// TIA Portal V17 export
// export: Created 2022-07-20T06:59:48.1085012Z, ExportSetting WithDefaults, DisplayName Totally Integrated Automation Portal, DisplayVersion V17, DisplayName TIA Portal Openness, DisplayVersion V17, DisplayName TIA Portal Version Control Interface, DisplayVersion V17, DisplayName SINAMICS Startdrive Advanced, DisplayVersion V17, DisplayName SINAMICS Startdrive G130, G150, S120, S150, SINAMICS MV, S210, DisplayVersion V17, DisplayName SINAMICS Startdrive G110M, G120, G120C, G120D, G120P, G115D, DisplayVersion V17, DisplayName STEP 7 Professional, DisplayVersion V17, DisplayName STEP 7 Safety, DisplayVersion V17, DisplayName WinCC Advanced, DisplayVersion V17
FUNCTION_BLOCK "FB10191_SheetTrackingProcess"   // FB10191, LAD
{ S7_Optimized_Access := 'TRUE' }
VERSION : 0.1
// stored: AutoNumber false, IsIECCheckEnabled false, IsRetainMemResEnabled false, MemoryReserve 100, SetENOAutomatically false, UDAEnableTagReadback false
   VAR_INPUT
      Enable : Bool;
      FirstSheetSensor : Bool;
      SecondSheetSensor : Bool;
      SheetSize : Real;   // mm
      TransportSpeed : Real;   // mm/s
      ActivationProcessMargin : Real;   // 0-100%
      DeactivationProcessMargin : Real;
      DistanceBetweenSheetSensors : Real;
      DistanceBetweenSheetSensorAndProcess : Real;
      RequestAcknowledge : Bool;
      Reset : Bool;
   END_VAR
   VAR_OUTPUT
      ActiveProcess : Bool;
      DeactiveProcess : Bool;
      TrackingProcessInError : Bool;
   END_VAR
   VAR
      i : SInt;
      R_TRIG_Enable : R_TRIG;
      R_TRIG_Reset { S7_SetPoint := 'True'} : R_TRIG;
      R_TRIG_Clock10Hz : R_TRIG;
      R_TRIG_SheetSensorSignal_1 { S7_SetPoint := 'True'} : R_TRIG;
      R_TRIG_SheetSensorSignal_2 { S7_SetPoint := 'True'} : R_TRIG;
      R_TRIG_SheetOutsideProcess { S7_SetPoint := 'True'} : R_TRIG;
      F_TRIG_Enable { S7_SetPoint := 'True'} : F_TRIG;
      F_TRIG_Clock10Hz { S7_SetPoint := 'True'} : F_TRIG;
      F_TRIG_SheetSensorSignal_1 { S7_SetPoint := 'True'} : F_TRIG;
      F_TRIG_SheetSensorSignal_2 { S7_SetPoint := 'True'} : F_TRIG;
      ARRAY_R_TRIGS_SheetsSensor_1 : Array[0..49] of Bool;
      ARRAY_R_TRIGS_SheetsSensor_2 : Array[0..49] of Bool;
      ARRAY_R_TRIGS_BeginningOfSheetUnderProcess : Array[0..49] of R_TRIG;
      ARRAY_R_TRIGS_EndOfSheetUnderProcess : Array[0..49] of R_TRIG;
      ARRAY_F_TRIGS_SheetsSensor_1 : Array[0..49] of Bool;
      ARRAY_F_TRIGS_SheetsSensor_2 : Array[0..49] of Bool;
      ARRAY_BeginingOfSheetPosition { S7_SetPoint := 'True'} : Array[0..49] of Real;   // mm
      ARRAY_EndOfSheetPosition { S7_SetPoint := 'True'} : Array[0..49] of Real;   // mm
      ARRAY_ElpasedTimeFromPreviousCheck { S7_SetPoint := 'True'} : Array[0..49] of Time;   // s
      ARRAY_TON_SheetsBetweenSensors : Array[0..49] of TON_TIME;
   END_VAR
BEGIN

REGION Network 1 (SCL): First Scan & Reset
   IF "FirstScan" OR #R_TRIG_Enable.Q OR #F_TRIG_Enable.Q OR #R_TRIG_Reset.Q THEN
       #ActiveProcess := FALSE;
       #DeactiveProcess := TRUE;
       FOR #i := 0 TO 49 DO
           #ARRAY_R_TRIGS_SheetsSensor_1[#i] := FALSE;
           #ARRAY_F_TRIGS_SheetsSensor_1[#i] := FALSE;
           #ARRAY_R_TRIGS_SheetsSensor_2[#i] := FALSE;
           #ARRAY_F_TRIGS_SheetsSensor_2[#i] := FALSE;
           #ARRAY_BeginingOfSheetPosition[#i] := 0.0;
           #ARRAY_EndOfSheetPosition[#i] := 0.0;
           #ARRAY_ElpasedTimeFromPreviousCheck[#i] := T#0s;
           RESET_TIMER(#ARRAY_TON_SheetsBetweenSensors[#i]);
       END_FOR;
   END_IF;
END_REGION

REGION Network 2 (SCL): Edge Signals & Timers
   REGION EDGE SIGNALS
       #R_TRIG_Enable(CLK := #Enable);
       #R_TRIG_Reset(CLK := #Reset);

       #F_TRIG_Enable(CLK := #Enable);
   END_REGION

   IF #Enable THEN
       REGION EDGE SIGNALS
           #R_TRIG_Clock10Hz(CLK := "Clock_10Hz");
           #R_TRIG_SheetSensorSignal_1(CLK := #FirstSheetSensor);
           #R_TRIG_SheetSensorSignal_2(CLK := #SecondSheetSensor);
           #R_TRIG_SheetOutsideProcess(CLK :=
                                       (#ARRAY_R_TRIGS_SheetsSensor_1[0] AND
                                       #ARRAY_R_TRIGS_SheetsSensor_2[0] AND
                                       #ARRAY_F_TRIGS_SheetsSensor_1[0] AND
                                       #ARRAY_F_TRIGS_SheetsSensor_2[0])
                                       OR
                                       (#ARRAY_BeginingOfSheetPosition[0] > 2 * #DistanceBetweenSheetSensors));

           #F_TRIG_Clock10Hz(CLK := "Clock_10Hz");
           #F_TRIG_SheetSensorSignal_1(CLK := #FirstSheetSensor);
           #F_TRIG_SheetSensorSignal_2(CLK := #SecondSheetSensor);

           FOR #i := 0 TO 49 DO
               #ARRAY_R_TRIGS_BeginningOfSheetUnderProcess[#i](CLK := #ARRAY_R_TRIGS_SheetsSensor_1[#i] AND "FC10021_TolerenceRelation"(X := #ARRAY_BeginingOfSheetPosition[#i], Y := #DistanceBetweenSheetSensorAndProcess, Tolerance := ((1 + #ActivationProcessMargin / 100) * 100)));
               #ARRAY_R_TRIGS_EndOfSheetUnderProcess[#i](CLK := #ARRAY_F_TRIGS_SheetsSensor_1[#i] AND "FC10021_TolerenceRelation"(X := #ARRAY_EndOfSheetPosition[#i], Y := #DistanceBetweenSheetSensorAndProcess, Tolerance := ((1 + #DeactivationProcessMargin / 100) * 100)));
           END_FOR;
       END_REGION

       REGION TIMERS
           FOR #i := 0 TO 49 DO
               #ARRAY_TON_SheetsBetweenSensors[#i](IN := #ARRAY_R_TRIGS_SheetsSensor_1[#i] AND NOT (#ARRAY_F_TRIGS_SheetsSensor_2[#i]),
                                                   PT := DINT_TO_TIME(REAL_TO_DINT((1 + (#ActivationProcessMargin / 100.0)) * (#DistanceBetweenSheetSensors / #TransportSpeed)) * 1000));
           END_FOR;
       END_REGION
   END_IF;
END_REGION

REGION Network 3 (SCL): Sheet Position Management
   IF #Enable THEN
      //Detect to Rising Edge of the first sensor
       IF #R_TRIG_SheetSensorSignal_1.Q THEN
           FOR #i := 0 TO 49 DO
               IF NOT (#ARRAY_R_TRIGS_SheetsSensor_1[#i]) THEN
                   #ARRAY_R_TRIGS_SheetsSensor_1[#i] := TRUE;
                   EXIT;
               END_IF;
           END_FOR;
       END_IF;

       //Detect the falling edge of the first sensor
       IF #F_TRIG_SheetSensorSignal_1.Q THEN
           FOR #i := 0 TO 49 DO
               IF #ARRAY_R_TRIGS_SheetsSensor_1[#i] AND NOT (#ARRAY_F_TRIGS_SheetsSensor_1[#i]) THEN
                   #ARRAY_F_TRIGS_SheetsSensor_1[#i] := TRUE;
                   EXIT;
               END_IF;
           END_FOR;
       END_IF;

       //Detect the rising edge of the second sensor
       IF #R_TRIG_SheetSensorSignal_2.Q THEN
           FOR #i := 0 TO 49 DO
               IF NOT (#ARRAY_R_TRIGS_SheetsSensor_2[#i]) AND "FC10021_TolerenceRelation"(X := #ARRAY_BeginingOfSheetPosition[#i], Y := #DistanceBetweenSheetSensors, Tolerance := 2000) THEN
                   #ARRAY_R_TRIGS_SheetsSensor_2[#i] := TRUE;
                   EXIT;
               END_IF;
           END_FOR;
       END_IF;

       //Detect the falling edge of the second sensor
       IF #F_TRIG_SheetSensorSignal_2.Q THEN
           FOR #i := 0 TO 49 DO
               IF #ARRAY_R_TRIGS_SheetsSensor_2[#i] AND NOT (#ARRAY_F_TRIGS_SheetsSensor_2[#i]) THEN
                   #ARRAY_F_TRIGS_SheetsSensor_2[#i] := TRUE;
                   EXIT;
               END_IF;
           END_FOR;
       END_IF;

       //Determine The Position Of The Beginning And The End Of The Sheet
       FOR #i := 0 TO 49 DO
           IF #ARRAY_R_TRIGS_SheetsSensor_1[#i] (*AND NOT (#ARRAY_R_TRIGS_SheetsSensor_2[#i])*)AND #R_TRIG_Clock10Hz.Q THEN
               #ARRAY_BeginingOfSheetPosition[#i] += (1 + #ActivationProcessMargin / 100) * (#TransportSpeed * 0.1);
           END_IF;

           IF #ARRAY_F_TRIGS_SheetsSensor_1[#i] (* AND NOT(#ARRAY_F_TRIGS_SheetsSensor_2[#i]) *)AND #R_TRIG_Clock10Hz.Q THEN
               #ARRAY_EndOfSheetPosition[#i] += (1 + #ActivationProcessMargin / 100) * (#TransportSpeed * 0.1);
           END_IF;
       END_FOR;

       IF #R_TRIG_SheetOutsideProcess.Q THEN
           FOR #i := 1 TO 49 DO
               #ARRAY_R_TRIGS_SheetsSensor_1[#i - 1] := #ARRAY_R_TRIGS_SheetsSensor_1[#i];
               #ARRAY_F_TRIGS_SheetsSensor_1[#i - 1] := #ARRAY_F_TRIGS_SheetsSensor_1[#i];
               #ARRAY_R_TRIGS_SheetsSensor_2[#i - 1] := #ARRAY_R_TRIGS_SheetsSensor_2[#i];
               #ARRAY_F_TRIGS_SheetsSensor_2[#i - 1] := #ARRAY_F_TRIGS_SheetsSensor_2[#i];
               #ARRAY_BeginingOfSheetPosition[#i - 1] := #ARRAY_BeginingOfSheetPosition[#i];
               #ARRAY_EndOfSheetPosition[#i - 1] := #ARRAY_EndOfSheetPosition[#i];
           END_FOR;
       END_IF;
   END_IF;
END_REGION

REGION Network 4 (SCL): Process Management
   IF #Enable THEN
       FOR #i := 0 TO 48 DO
           IF #ARRAY_R_TRIGS_BeginningOfSheetUnderProcess[#i].Q AND NOT (#ActiveProcess) THEN
               #ActiveProcess := TRUE;
               #DeactiveProcess := FALSE;
           END_IF;

           IF
               (#ARRAY_R_TRIGS_EndOfSheetUnderProcess[#i].Q AND
               NOT (#ARRAY_R_TRIGS_SheetsSensor_1[#i + 1]) AND
               #ActiveProcess)
               OR
               (#ARRAY_BeginingOfSheetPosition[0] = 0.0 AND
               #ARRAY_EndOfSheetPosition[0] = 0.0)
           THEN
               #ActiveProcess := FALSE;
               #DeactiveProcess := TRUE;
           END_IF;
       END_FOR;
   ELSE
       #ActiveProcess := FALSE;
       #DeactiveProcess := TRUE;
   END_IF;
END_REGION

REGION Network 5 (SCL): Error Management
   //Sheet Tracking Process Error Management
   IF #ARRAY_BeginingOfSheetPosition[49] > 0.0 THEN
       #TrackingProcessInError := TRUE;
   END_IF;

   //Acknowledge Management
   IF #RequestAcknowledge THEN
       #TrackingProcessInError := FALSE;
   END_IF;
END_REGION
END_FUNCTION_BLOCK
